Universal Robots PolyScope program: g_to_d.urp

Program g_to_d (installation=string_planes directory=/programs/string_crossings createdIn=5.17.3 lastSavedIn=5.17.3 robotSerialNumber=20245501435)
Calibrated DH parameters: a=[0.000154, -0.137004, -0.385524, -0.00002, 0.000092, 0]; d=[0.162441, 211.794786, -230.585024, 18.923638, 0.099786, 0.09951]; alpha=[1.569493, -0.001902, 0.003874, 1.570111, -1.570167, 0]; deltaTheta=[0, -1.242934, 1.056292, 0.186646, 0.000002, 0.000001]
InitVariablesNode
Robot Program (runOnlyOnce=true)
  bow_section := -1
  If bow_section≟-1
    MoveJ speed 60 deg/s, acceleration 80 deg/s^2 (useActiveTCP=true) feature=Base
      Waypoint Waypoint_2 (Relative): relativeFromPosition TCP in base x=333.345 y=655.475 z=103.654 mm, rx=-1.6491 ry=-1.7982 rz=0.6656 rad; joints [-132.466, -27.757, 71.843, -100.482, -56.044, -147.73] deg; TCP offset x=28.21 y=-96.107 z=-99.69 mm, rx=0 ry=0 rz=0 rad; TCP in base x=316.098 y=723.605 z=117.805 mm, rx=-1.5349 ry=-2.2386 rz=1.1275 rad; joints [-128.46, -21.869, 50.821, -72.93, -81.955, -152.853] deg
  ElseIf bow_section≟0
    MoveJ speed 60 deg/s, acceleration 80 deg/s^2 (useActiveTCP=true) feature=Base
      Waypoint Waypoint_1 (Relative): relativeFromPosition TCP in base x=267.758 y=455.827 z=63.35 mm, rx=-1.6064 ry=-1.9107 rz=0.8702 rad; joints [-141.614, -39.193, 108.913, -115.288, -70.78, -159.119] deg; TCP in base x=337.277 y=452.587 z=146.27 mm, rx=-1.6083 ry=-2.1978 rz=1.0429 rad; joints [-146.227, -47.168, 100.748, -99.801, -91.438, -163.024] deg
  Else 
    MoveJ speed 60 deg/s, acceleration 80 deg/s^2 (useActiveTCP=true) feature=Base
      Waypoint Waypoint_3 (Relative): relativeFromPosition TCP in base x=243.623 y=214.066 z=64.413 mm, rx=-1.5874 ry=-1.9212 rz=0.962 rad; joints [-169.308, -44.603, 138.124, -133.881, -94.42, -177.776] deg; TCP in base x=340.792 y=238.623 z=127.333 mm, rx=-1.5375 ry=-2.1223 rz=1.0864 rad; joints [-167.854, -53.469, 123.57, -113.681, -104.544, -179.466] deg
